{attribute addProperty BoxType "EL9560-0000-0016"}
{attribute addProperty Id "Power_OKAT %I*BOOL81"}
{attribute addProperty CRC "843727106"}
{attribute addProperty SizeInBites "8"}
{attribute addProperty SizeInBytes "1"}
TYPE Status_Us_324A4102 :
STRUCT
	{attribute addProperty Name "Power_OK"}
	Power_OK AT %I* : BOOL;
END_STRUCT
END_TYPE

(* stored: Version 1.2.0.0, ProductVersion 3.1.4024.9
   DUT Status_Us_324A4102: Id {a305367e-2cc0-42d6-af04-050b428e1a11} *)
